(* CODESYS project OC_Core.library
   DefaultNamespace: OC_Core
   DocFormat: reStructuredText
   Description: Open Commissioning TwinCAT Core Library
   Author: SpiraTec AG
   Title: OC_Core
   Version: 1.3.1
   Company: Open Commissioning
   Placeholder: OC_Core

Project tree, tasks and I/O mapping:
  libraries: Tc2_Math, 3.4.4.0 (Beckhoff Automation GmbH); Tc2_Standard, 3.4.5.0 (Beckhoff Automation GmbH); Tc2_System, 3.6.4.0 (Beckhoff Automation GmbH); Tc2_Utilities, 3.6.1.0 (Beckhoff Automation GmbH); Tc3_Module, 3.4.5.0 (Beckhoff Automation GmbH); TcUnit, 1.3.0.0 (www.tcunit.org)
  Common/
    AdsMessageHandler/
      function block FB_AdsMessageHandler [ST]: bIsAdsMessageReadValid, bIsAdsMessageWriteValid, CreateAdsReadMessage, CreateAdsWriteMessage, LogAdsMessage, SendReadResponse, SendWriteResponse, stAdsMessageRead, stAdsMessageWrite
      data type ST_AdsMessage
    Components/
      Encoder/
        function block FB_Encoder [ST]: ControlLogic, INC_TO_LREAL, InitRun, LREAL_TO_INC, SetActualValue
        data type ST_Encoder_Config
      function block FB_Clock [ST]
      function block FB_ClockAdvanced [ST]
      function block FB_DriveControl [ST]: bIsMoving, bIsPositionReached, fAccMax, fPosition, fPositionLimitMax, fPositionLimitMin, fTolerance, fVelocity, MoveAbsolute, MoveVelocity, Stop
      function block FB_Heater [ST]: fValue, InitRun
      function block FB_MoveAbsolute [ST]: bIsReached, fPosition, fVelocity
      function block FB_MoveVelocity [ST]: bIsReached, fAcc, fVelocity
      function block FB_Ping [ST]: InitRun
    FileIo/
      data type E_FileIoState
      function block FB_FileIO [ST]: nBytesRead, nErrorId, Read, sNetId, Write
    Links/
      function block FB_LinkDataByte [ST]: GetLinkControlData, SetLinkStatusData
      function block FB_LinkDataDWord [ST]: GetLinkControlData, SetLinkStatusData
      function block FB_LinkDataLWord [ST]: GetLinkControlData, SetLinkStatusData
      function block FB_LinkDataReal [ST]: GetLinkControlData, SetLinkStatusData
      function block FB_LinkDataWord [ST]: GetLinkControlData, SetLinkStatusData
      function block FB_LinkDevice [ST]: GetControl, SetStatus
    RecordData/
      function block FB_RecordData [ST]: CmpIGrp, CmpInvokeId, CmpIOffs, DataValid, FB_init, GetReadIndication, GetWriteIndication, SendReadResponse, SendWriteResponse, Subscribe
      interface I_RecordData: GetReadIndication, GetWriteIndication, SendReadResponse, SendWriteResponse, Subscribe
      data type ST_RecordIdent
    System/
      data type E_ControllerType
      function F_IsSystemValid [ST]
      function F_LogError [ST]
      function F_LogMessage [ST]
      function F_LogWarning [ST]
      function block FB_Base [ST]
      function block FB_System [ST]: bDebug, bVerbose, eControllerType, fDeltaTime, fTimeScaling, InitRun
      global variables GVL_Core
    Utils/
      data type E_NetworkByteOrder
      function F_Clamp01 [ST]
      function F_Compare [ST]
      function F_GetHByte [ST]
      function F_GetLByte [ST]
      function F_InverBytesOrder [ST]
      function F_Memcpy [ST]
      function F_Norm [ST]
      function F_ScaleLREAL [ST]
      function F_Sign [ST]
      data type ST_ScaleConfig
  Devices/
    Basic/
      function block FB_Button [ST]
      function block FB_Cylinder [ST]
      function block FB_Device [ST]
      function block FB_DeviceByte [ST]
      function block FB_DeviceDWord [ST]
      function block FB_DeviceLWord [ST]
      function block FB_DeviceReal [ST]
      function block FB_DeviceWord [ST]
      function block FB_Drive [ST]
      function block FB_Lamp [ST]
      function block FB_Lock [ST]
      function block FB_Panel [ST]
      function block FB_Reader [ST]
      function block FB_Robot [ST]: ConnectJoints, GetJointsTarget, SetJointsStatus
      function block FB_SensorAnalog [ST]
      function block FB_SensorBinary [ST]
      function block FB_Switch [ST]
*)

// Common/AdsMessageHandler/ST_AdsMessage
TYPE ST_AdsMessage :
STRUCT
	tNetID			: T_AmsNetID; // AMS NetId identifier
	tPort			: T_AmsPort; // AMS port number
	nInvokeID		: UDINT; // Unique identifier for the ADS invocation
	nIdxGrp			: UDINT; // Index group for the ADS command
	nIdxOffs		: UDINT; // Index offset within the ADS command
	nLength			: UDINT; // Length of the ADS message data
	nResult			: UDINT; // Result code from the ADS operation
	aData			: ARRAY[0..239] OF BYTE; // Data payload (240-byte buffer)
END_STRUCT
END_TYPE

// Common/Components/Encoder/ST_Encoder_Config
TYPE ST_Encoder_Config :
STRUCT
	bIsIntegrator   		: BOOL := FALSE;  //Integrate input value
	fNumerator 	  			: REAL := 0.0001; //[unit/INC]
	fDenominator  			: REAL := 1.0; 	// Scaling
	fModulo 	  			: REAL := 0; // Modulo [unit]; If 0, will be ignored
	fGearFactor  			: REAL := 1.0;
	bInvertEncoderDirection : BOOL;
END_STRUCT
END_TYPE

// Common/FileIo/E_FileIoState
{attribute 'conditionalshow'}
TYPE E_FileIoState :
(
	READY := 0,
	OPEN,
	CREATE,
	READ,
	WRITE,
	CLOSE,
	ERROR
);
END_TYPE

// Common/RecordData/ST_RecordIdent
TYPE ST_RecordIdent :
STRUCT
	nPort  			: T_AmsPort; //ADS-Port of the Profinet Device. Ignored when using PLCSIM Advanced
	nSlot			: UINT; //Slotnumber of the Profinet Device. Ignored when using PLCSIM Advanced
	nSubSlot		: UINT; //Subslotnumber of the Profinet Device. Ignored when using PLCSIM Advanced
	nPlcId			: UINT; //Identifier of the PLC when using PLCSIM Advanced
	nHardwareId		: UINT; //Hardware-ID of the device when using PLCSIM Advanced
END_STRUCT
END_TYPE

// Common/System/E_ControllerType
{attribute 'qualified_only'}
{attribute 'strict'}
TYPE E_ControllerType :
(
	NotDefined := 0,
	PlcSimAdvanced := 1
);
END_TYPE

// Common/Utils/E_NetworkByteOrder
{attribute 'qualified_only'}
{attribute 'strict'}
TYPE E_NetworkByteOrder :
(
	BigEndian := 0, //Big Endian (MOTOROLA)
	LittleEndian := 1 //Little Endian (Intel)	
);
END_TYPE

// Common/Utils/ST_ScaleConfig
{attribute 'pack_mode' := '0'} 
TYPE ST_ScaleConfig :
STRUCT
	fInputMin 	: LREAL := 0;
	fInputMax 	: LREAL := 100;
	fOutputMin 	: LREAL := 0;
	fOutputMax 	: LREAL := 65535;
END_STRUCT
END_TYPE

// Common/System/GVL_Core
{attribute 'qualified_only'}
{attribute 'conditionalshow'}
VAR_GLOBAL	
	refSystem 			: REFERENCE TO FB_System;		
END_VAR

// Common/AdsMessageHandler/FB_AdsMessageHandler
(*ADS Message Handler is responsible for indication of the ADS Read/Write messages for local NetId and generation of the response message*)
FUNCTION_BLOCK FB_AdsMessageHandler
VAR_INPUT
	bDisable 				: BOOL;	//Deactivate cyclical execution
	bLog					: BOOL;	//Log ADS messages data in the console
	bVerbose				: BOOL; //Log Verbose information in the console
END_VAR

VAR	
	_fbAdsWriteIndicator 	: AdsWriteInd;	
	_fbAdsReadIndicator 	: AdsReadInd;
	_fbAdsWriteResponse		: AdsWriteRes;
	_fbAdsReadResponse		: AdsReadRes;	
	_stAdsMessageWrite		: ST_AdsMessage;
	_stAdsMessageRead		: ST_AdsMessage;
END_VAR

VAR CONSTANT
	S_FORMAT_RECEIVEWRITE	: STRING := 'AdsWriteInd Port: %X, IdxGrp: %X, IdxOffs: %X, InvokeId %X, Length: %X';
	S_FORMAT_RECEIVEREAD	: STRING := 'AdsReadInd Port: %X, IdxGrp: %X, IdxOffs: %X, InvokeId %X, Length: %X';
	S_FORMAT_RESPONSEWRITE	: STRING := 'AdsWriteRes Port: %X, IdxGrp: %X, IdxOffs: %X, InvokeId %X, Length: %X';
	S_FORMAT_RESPONSEREAD	: STRING := 'AdsReadRes Port: %X, IdxGrp: %X, IdxOffs: %X, InvokeId %X, Length: %X';  
END_VAR

IF bDisable THEN RETURN; END_IF

//Reset Indication and Result FBs
_fbAdsWriteResponse(RESPOND := FALSE);
_fbAdsReadResponse(RESPOND := FALSE);

//Capture all Write requests
_fbAdsWriteIndicator();
CreateAdsWriteMessage();
		
//Capture all Read requests
_fbAdsReadIndicator();
CreateAdsReadMessage();

(*Returns the status of the indication of the read message in the current frame*)
PROPERTY PUBLIC bIsAdsMessageReadValid : BOOL
GET
bIsAdsMessageReadValid := _stAdsMessageRead.tPort <> 0;
END_GET
END_PROPERTY

(*Returns the status of the indication of the write message in the current frame*)
PROPERTY PUBLIC bIsAdsMessageWriteValid : BOOL
GET
bIsAdsMessageWriteValid := _stAdsMessageWrite.tPort <> 0;
END_GET
END_PROPERTY

METHOD PRIVATE CreateAdsReadMessage : BOOL
IF NOT _fbAdsReadIndicator.VALID THEN RETURN; END_IF

MEMSET(ADR(_stAdsMessageRead), 0, SIZEOF(ST_AdsMessage));
_stAdsMessageRead.tNetId 		:= _fbAdsReadIndicator.NETID;
_stAdsMessageRead.tPort 		:= _fbAdsReadIndicator.PORT;
_stAdsMessageRead.nInvokeId 	:= _fbAdsReadIndicator.INVOKEID;
_stAdsMessageRead.nIdxGrp 		:= _fbAdsReadIndicator.IDXGRP;
_stAdsMessageRead.nIdxOffs 		:= _fbAdsReadIndicator.IDXOFFS;
_stAdsMessageRead.nLength 		:= _fbAdsReadIndicator.LENGTH;

IF bVerbose THEN
	LogAdsMessage(_stAdsMessageWrite, S_FORMAT_RECEIVEREAD);
END_IF

_fbAdsReadIndicator(CLEAR := TRUE);
_fbAdsReadIndicator(CLEAR := FALSE);
END_METHOD

METHOD PRIVATE CreateAdsWriteMessage : BOOL
IF NOT _fbAdsWriteIndicator.VALID THEN RETURN; END_IF

MEMSET(ADR(_stAdsMessageWrite), 0, SIZEOF(ST_AdsMessage));
_stAdsMessageWrite.tNetId 		:= _fbAdsWriteIndicator.NETID;
_stAdsMessageWrite.tPort 		:= _fbAdsWriteIndicator.PORT;
_stAdsMessageWrite.nInvokeId 	:= _fbAdsWriteIndicator.INVOKEID;
_stAdsMessageWrite.nIdxGrp 		:= _fbAdsWriteIndicator.IDXGRP;
_stAdsMessageWrite.nIdxOffs 	:= _fbAdsWriteIndicator.IDXOFFS;
_stAdsMessageWrite.nLength 		:= _fbAdsWriteIndicator.LENGTH;
			
//Limit size to 240
IF _stAdsMessageWrite.nLength > 240 THEN
	IF bVerbose THEN
		F_LOGWARNING(CONCAT('WRREC data length limited to 240. Requested data length was ', TO_STRING(_stAdsMessageWrite.nLength)));
	END_IF
	_stAdsMessageWrite.nLength := 240;
END_IF

MEMCPY(ADR(_stAdsMessageWrite.aData), _fbAdsWriteIndicator.DATAADDR, _stAdsMessageWrite.nLength);

IF bVerbose THEN
	LogAdsMessage(_stAdsMessageWrite, S_FORMAT_RECEIVEWRITE);
END_IF

_fbAdsWriteIndicator(CLEAR := TRUE);
_fbAdsWriteIndicator(CLEAR := FALSE);
END_METHOD

METHOD PRIVATE LogAdsMessage : BOOL
VAR_INPUT
	stAdsMessage 			: ST_AdsMessage;
	sFormat 				: STRING;
END_VAR

VAR
	fbFormatString			: FB_FormatString2;
	sMessage				: STRING;
END_VAR
fbFormatString(
	pFormatString := ADR(sFormat),
	arg1 := F_UINT(stAdsMessage.tPort),
	arg2 := F_UDINT(stAdsMessage.nIdxGrp),
	arg3 := F_UDINT(stAdsMessage.nIdxOffs),		
	arg4 := F_UDINT(stAdsMessage.nInvokeID),
	arg5 := F_UDINT(stAdsMessage.nLength),
	pDstString := ADR(sMessage),
	nDstSize := SIZEOF(sMessage));
F_LogMessage(sMessage);
END_METHOD

(*Send ADS Read Response message*)
METHOD PUBLIC SendReadResponse : HRESULT
VAR_INPUT
	stAdsMessage 	: ST_AdsMessage; //Response ADS Message
END_VAR
IF _fbAdsReadResponse.RESPOND THEN
	SendReadResponse := S_PENDING;
	RETURN;
END_IF

//Limit size to 240
IF stAdsMessage.nLength > 240 THEN
	IF bVerbose THEN
		F_LOGWARNING(CONCAT('RDRES data length limited to 240. Requested data length was ', TO_STRING(stAdsMessage.nLength)));
	END_IF
	stAdsMessage.nLength := 240;
END_IF

_fbAdsReadResponse(
	NETID:= stAdsMessage.tNetId, 
	PORT:= stAdsMessage.tPort, 
	INVOKEID:= stAdsMessage.nInvokeId, 
	RESULT:= stAdsMessage.nResult, 
	LEN:= stAdsMessage.nLength,
	DATAADDR:= ADR(stAdsMessage.aData),
	RESPOND:= TRUE);
IF bVerbose OR bLog THEN	
	LogAdsMessage(stAdsMessage, S_FORMAT_RESPONSEREAD);
END_IF

SendReadResponse := S_OK;
END_METHOD

(*Send ADS Write Response message*)
METHOD PUBLIC SendWriteResponse : HRESULT
VAR_INPUT
	stAdsMessage 	: ST_AdsMessage; //Response ADS Message
END_VAR
IF _fbAdsWriteResponse.RESPOND THEN
	SendWriteResponse := S_PENDING;
	RETURN;
END_IF

_fbAdsWriteResponse(
	NETID:= stAdsMessage.tNetId, 
	PORT:= stAdsMessage.tPort, 
	INVOKEID:= stAdsMessage.nInvokeId, 
	RESULT:= stAdsMessage.nResult, 
	RESPOND:= TRUE);	

IF bVerbose OR bLog THEN		
	LogAdsMessage(stAdsMessage, S_FORMAT_RESPONSEWRITE);
END_IF
	
SendWriteResponse := S_OK;
END_METHOD

(*Get last valid ADS Read Message*)
PROPERTY stAdsMessageRead : REFERENCE TO ST_AdsMessage
GET
stAdsMessageRead REF= _stAdsMessageRead;
END_GET
END_PROPERTY

(*Get last valid ADS Write Message*)
PROPERTY stAdsMessageWrite : REFERENCE TO ST_AdsMessage
GET
stAdsMessageWrite REF= _stAdsMessageWrite;
END_GET
END_PROPERTY

END_FUNCTION_BLOCK

// Common/System/F_LogWarning
(*
	Log Warning message to TwinCAT console
*)
{attribute 'hide_all_locals'}
FUNCTION F_LogWarning : BOOL
VAR_INPUT
	sMessage : T_MAXSTRING;
END_VAR

VAR CONSTANT	
	S_LOGHEADER		: T_MAXSTRING := 'Open Commissioning: %s';
END_VAR

ADSLOGSTR(ADSLOG_MSGTYPE_WARN, S_LOGHEADER, sMessage);

END_FUNCTION

// Common/System/F_LogMessage
(*
	Log message to TwinCAT console
*)
{attribute 'hide_all_locals'}
FUNCTION F_LogMessage : BOOL
VAR_INPUT
	sMessage : T_MAXSTRING;
END_VAR

VAR CONSTANT	
	S_LOGHEADER		: T_MAXSTRING := 'Open Commissioning: %s';
END_VAR

ADSLOGSTR(ADSLOG_MSGTYPE_HINT, S_LOGHEADER, sMessage);

END_FUNCTION

// Common/Components/Encoder/FB_Encoder
(*
	Generic simulated Encoder 
*)
{attribute 'reflection'} 
FUNCTION_BLOCK FB_Encoder
VAR_INPUT
	fValue 			: LREAL; //Input Value [unit] or [unit/s]	
	stConfig 		: ST_Encoder_Config;	
END_VAR

VAR_OUTPUT
	nResult 		: DINT; //Position [INC]
	fResult 		: LREAL;
END_VAR

VAR
	{attribute 'instance-path'} 
    {attribute 'noinit'} 
    _sPath 				: STRING;
	_fValue 			: LREAL;
END_VAR

InitRun();
ControlLogic();

METHOD PRIVATE ControlLogic
IF stConfig.bIsIntegrator THEN
	_fValue := _fValue + (fValue * stConfig.fGearFactor * GVL_Core.fbSystem.fDeltaTime);
ELSE
	_fValue := fValue * stConfig.fGearFactor;
END_IF

IF stConfig.fModulo > 0.0 THEN
	_fValue := LREAL_TO_REAL(LMOD(_fValue, stConfig.fModulo));
END_IF

fResult := _fValue;

IF stConfig.bInvertEncoderDirection THEN
	nResult := LREAL_TO_INC(fResult, -1);
ELSE
	nResult := LREAL_TO_INC(fResult, 1);	
END_IF
END_METHOD

METHOD INC_TO_LREAL : LREAL
VAR_INPUT
	nValue : DINT;
	fFactor : LREAL;
END_VAR
//Parameters validation
stConfig.fNumerator := MAX(1E-6, stConfig.fNumerator);
stConfig.fDenominator := MAX(1E-6, stConfig.fDenominator);

INC_TO_LREAL := DINT_TO_REAL(nValue) * (stConfig.fNumerator / stConfig.fDenominator) * fFactor;
END_METHOD

METHOD PRIVATE InitRun
VAR_INST
	bInitRun : BOOL := TRUE;
END_VAR
IF NOT bInitRun THEN RETURN; END_IF
bInitRun := FALSE;
END_METHOD

METHOD LREAL_TO_INC : DINT
VAR_INPUT
	fValue : LREAL;
	fFactor : LREAL;
END_VAR
//Parameters validation
stConfig.fNumerator := MAX(1E-6, stConfig.fNumerator);
stConfig.fDenominator := MAX(1E-6, stConfig.fDenominator);

LREAL_TO_INC := LREAL_TO_DINT(fValue * (stConfig.fDenominator / stConfig.fNumerator) * fFactor);
END_METHOD

METHOD PUBLIC SetActualValue : BOOL
VAR_INPUT
	fValue : LREAL;
END_VAR
_fValue := fValue;
END_METHOD

END_FUNCTION_BLOCK

// Common/Components/FB_Clock
FUNCTION_BLOCK FB_Clock
VAR_INPUT
	tPT		: TIME;
END_VAR

VAR_OUTPUT
	bQ		: BOOL;
END_VAR

VAR
	_fbTon1	: TON;
	_fbTon2	: TON;
END_VAR

_fbTon1.PT := tPT;
_fbTon2.PT := tPT;

_fbTon1(IN := NOT bQ);
_fbTon2(IN := bQ);

IF _fbTon1.Q THEN
	bQ := TRUE;
END_IF

IF _fbTon2.Q THEN
	bQ := FALSE;
END_IF

END_FUNCTION_BLOCK

// Common/Components/FB_ClockAdvanced
FUNCTION_BLOCK FB_ClockAdvanced
VAR_INPUT
	bEnable				: BOOL;
	tImpulsePTHigh		: TIME;
	tImpulsePTLow		: TIME;
	tDelay				: TIME;
	bInvert				: BOOL;
END_VAR

VAR_OUTPUT
	bQ					: BOOL;
END_VAR

VAR
	_fbTon1				: TON;
	_fbTon2				: TON;
	_fbTonDelay 		: TON;
	_bValue 			: BOOL;
END_VAR

_fbTonDelay.IN := bEnable;
_fbTonDelay.PT := tDelay;
_fbTonDelay();

IF NOT bEnable THEN
	bQ := FALSE;
	_fbTon1(IN := FALSE);
	_fbTon2(IN := FALSE);
	RETURN;
END_IF

IF _fbTonDelay.Q THEN
	IF bInvert THEN
		_fbTon1.PT := tImpulsePTHigh;
		_fbTon2.PT := tImpulsePTLow;
	ELSE
		_fbTon1.PT := tImpulsePTLow;
		_fbTon2.PT := tImpulsePTHigh;
	END_IF
	
	_fbTon1(IN := NOT _bValue);
	_fbTon2(IN := _bValue);
	
	IF _fbTon1.Q THEN
		_bValue := TRUE;
	END_IF
	
	IF _fbTon2.Q THEN
		_bValue := FALSE;
	END_IF	
	
	IF bInvert THEN
		bQ := NOT _bValue;
	ELSE
		bQ := _bValue;	
	END_IF	
END_IF

END_FUNCTION_BLOCK

// Common/Components/FB_DriveControl
(*
	FB_DriveControl manages drive operations by integrating absolute position and velocity control.
    It encapsulates the functionalities of FB_MoveAbsolute for absolute movement and FB_MoveVelocity
    for velocity-based control.
*)
FUNCTION_BLOCK FB_DriveControl
VAR
	_fbMoveAbsolute 		: FB_MoveAbsolute();
	_fbMoveVelocity			: FB_MoveVelocity();

	_fPosition 				: REAL;
	_fVelocity 				: REAL;		
	_bIsPositionReached 	: BOOL := TRUE;		
	
	_fPositionLimitMin 		: REAL := -1E+12;
	_fPositionLimitMax 		: REAL := 1E+12;
	_fAccMax				: REAL := 1E+12;	
	_fTolerance				: REAL := 1E-6;	
END_VAR

(*
    Indicates whether the drive is currently in motion.

    The bIsMoving property returns TRUE if the drive is actively moving toward its target.
*)
PROPERTY bIsMoving : BOOL
GET
bIsMoving := NOT F_Compare(_fVelocity, 0, 1E-3);
END_GET
END_PROPERTY

(*
    Indicates whether the drive has reached its target position.

    This property reflects the internal state of the drive control system.
    It returns TRUE if the drive has achieved the desired position within the specified
    tolerance limits; otherwise, it returns FALSE.
*)
PROPERTY bIsPositionReached : BOOL
GET
bIsPositionReached := _bIsPositionReached;
END_GET
END_PROPERTY

(*
    Maximum Acceleration Limit

    The fAccMax property represents the maximum acceleration permitted for drive movements.
*)
PROPERTY fAccMax : REAL
GET
fAccMax := _fAccMax;
END_GET
SET
_fAccMax := fAccMax;
END_SET
END_PROPERTY

(*
    Actual Drive Position
	
	The fPosition property provides the current position for the drive.
*)
PROPERTY fPosition : REAL
GET
fPosition := _fPosition;
END_GET
SET
_fPosition := fPosition;
END_SET
END_PROPERTY

(*
    Maximum Position Limit
	
	The fPositionLimitMax property defines the upper boundary for the drive's position.
*)
PROPERTY fPositionLimitMax : REAL
GET
fPositionLimitMax := _fPositionLimitMax;
END_GET
SET
_fPositionLimitMax := fPositionLimitMax;
END_SET
END_PROPERTY

(*
    Minimum  Position Limit
	
	The fPositionLimitMax property defines the lower boundary for the drive's position.
*)
PROPERTY fPositionLimitMin : REAL
GET
fPositionLimitMin := _fPositionLimitMin;
END_GET
SET
_fPositionLimitMin := fPositionLimitMin;
END_SET
END_PROPERTY

(*
    Position Tolerance
	
	The fTolerance property defines the acceptable error range for the drive's position.
*)
PROPERTY fTolerance : REAL
GET
fTolerance := _fTolerance;
END_GET
SET
_fTolerance := fTolerance;
END_SET
END_PROPERTY

(*
    Actual Drive Velocity
	
	The fVelocity property provides the current velocity for the drive.
*)
PROPERTY fVelocity : REAL
GET
fVelocity := _fVelocity;
END_GET
SET
_fVelocity := fVelocity;
END_SET
END_PROPERTY

(* 
    Moves the drive to an absolute position.
    
    The MoveAbsolute method commands the drive to move to a specified absolute position with a given velocity,
    acceleration, and deceleration.
*)
METHOD MoveAbsolute
VAR_INPUT
	fPosition 			: REAL;
	fVelocity			: REAL;
	fAcceleration		: REAL;
	fDeceleration   	: REAL;
END_VAR
_fbMoveAbsolute.fPosition := _fPosition;
_fbMoveAbsolute.fVelocity := _fVelocity;

_fbMoveAbsolute(
	fTargetPosition := LIMIT(_fPositionLimitMin, fPosition, _fPositionLimitMax),
	fTargetVelocity := fVelocity,
	fAccMax := fAcceleration,
	fDecMax := fDeceleration,
	fTolerance := _fTolerance);					

_fVelocity := _fbMoveAbsolute.fVelocity;
_fPosition := _fbMoveAbsolute.fPosition;

_bIsPositionReached := F_Compare(fPosition, _fPosition, _fTolerance);
END_METHOD

(* 
    Moves the drive using velocity control.
    
    The MoveVelocity method commands the drive to move with a specified velocity and controls the acceleration
    and deceleration parameters. It also enforces position limits to prevent the drive from exceeding its boundaries.
*)
METHOD MoveVelocity
VAR_INPUT
	fVelocity 			: REAL;
	fAcceleration 		: REAL;
	fDeceleration 		: REAL;
END_VAR
_fbMoveVelocity.fVelocity := _fVelocity;
_fbMoveVelocity.fTargetVelocity := fVelocity;
_fbMoveVelocity.fAccMax := fAcceleration;
_fbMoveVelocity.fDecMax := fDeceleration;	
	
IF _fPositionLimitMax <> 0 AND _fPositionLimitMin <> 0 THEN
	IF _fPosition >= _fPositionLimitMax OR _fPosition <= _fPositionLimitMin THEN
		_fbMoveVelocity.fTargetVelocity := 0;
		_fbMoveVelocity.fAccMax := _fAccMax;
		_fbMoveVelocity.fDecMax := _fAccMax;
	END_IF		
END_IF
	
_fbMoveVelocity();
	
_fVelocity := _fbMoveVelocity.fVelocity;	

_fPosition := _fPosition + _fVelocity * GVL_Core.fbSystem.fDeltaTime * GVL_Core.fbSystem.fTimeScaling;
_bIsPositionReached := F_Compare(fPosition, _fPosition, _fTolerance);
END_METHOD

(* 
    Stops the drive movement.
    
    The Stop method decelerates the drive until it comes to a complete halt using the specified deceleration.
*)
METHOD Stop
VAR_INPUT
	fDeceleration 	: REAL; 
END_VAR

VAR
	fSign 			: REAL;
	fAbsVelocity 	: REAL;
END_VAR
fSign := F_Sign(_fVelocity);
fAbsVelocity := ABS(_fVelocity);

IF fAbsVelocity > fTolerance THEN
	fAbsVelocity := fAbsVelocity - ABS(fDeceleration) * GVL_Core.fbSystem.fDeltaTime * GVL_Core.fbSystem.fTimeScaling;
	fAbsVelocity := LIMIT(0, fAbsVelocity, 3.402823E+38);
	_fVelocity := fAbsVelocity * fSign;	
ELSE
	_fVelocity := 0;
END_IF
END_METHOD

END_FUNCTION_BLOCK

// Common/Components/FB_MoveAbsolute
(* 
	FB_MoveAbsolute: Controls absolute movement using target position, velocity, acceleration, and deceleration. 
*)
FUNCTION_BLOCK FB_MoveAbsolute 
VAR_INPUT
	fTargetPosition 	: REAL;
	fTargetVelocity 	: REAL; 
	fAccMax 			: REAL; 
	fDecMax 			: REAL;	
	fTolerance			: REAL := 1E-6;	
END_VAR

VAR
	_fVelocity 			: REAL;
	_fPosition 			: REAL;
	_bIsReached			: BOOL;
END_VAR

fTargetVelocity := ABS(fTargetVelocity); 
fAccMax := ABS(fAccMax);
fDecMax := -ABS(fDecMax);

IF F_Compare(fTargetPosition, _fPosition, fTolerance) THEN
	_fVelocity := 0;
	_fPosition := fTargetPosition;
	_bIsReached := TRUE;	
ELSE
	(* Calculate velocity and position *)
	IF fTargetPosition > _fPosition THEN		
		IF _fVelocity < 0 THEN
			_fVelocity := MIN(_fVelocity - fDecMax * GVL_Core.fbSystem.fDeltaTime * GVL_Core.fbSystem.fTimeScaling, fTargetVelocity);
		ELSE
			IF _fVelocity > fTargetVelocity THEN
				_fVelocity := MAX(_fVelocity + fDecMax * GVL_Core.fbSystem.fDeltaTime * GVL_Core.fbSystem.fTimeScaling, fTargetVelocity);
			ELSE
				_fVelocity := MIN(_fVelocity + fAccMax * GVL_Core.fbSystem.fDeltaTime * GVL_Core.fbSystem.fTimeScaling, fTargetVelocity);
			END_IF

			_fVelocity := MIN(SQRT((_fPosition - fTargetPosition) * 2.0 * fDecMax - 1.5 * GVL_Core.fbSystem.fDeltaTime * GVL_Core.fbSystem.fTimeScaling * fDecMax), _fVelocity);
		END_IF

		_fPosition := _fPosition + MIN(_fVelocity * GVL_Core.fbSystem.fDeltaTime * GVL_Core.fbSystem.fTimeScaling, fTargetPosition - _fPosition);	
	ELSE		
		IF _fVelocity > 0 THEN
			_fVelocity := MAX(_fVelocity + fDecMax * GVL_Core.fbSystem.fDeltaTime * GVL_Core.fbSystem.fTimeScaling, -fTargetVelocity);
		ELSE
			IF _fVelocity < -fTargetVelocity THEN
				_fVelocity := MIN(_fVelocity - fDecMax * GVL_Core.fbSystem.fDeltaTime * GVL_Core.fbSystem.fTimeScaling, -fTargetVelocity);
			ELSE				
				_fVelocity := MAX(_fVelocity - fAccMax * GVL_Core.fbSystem.fDeltaTime * GVL_Core.fbSystem.fTimeScaling, -fTargetVelocity);
			END_IF
			
			_fVelocity := MAX(-SQRT((_fPosition - fTargetPosition) * 2.0 * -fDecMax - 1.5 * GVL_Core.fbSystem.fDeltaTime * GVL_Core.fbSystem.fTimeScaling * fDecMax), _fVelocity);
	   END_IF

		_fPosition := _fPosition + MAX(_fVelocity * GVL_Core.fbSystem.fDeltaTime * GVL_Core.fbSystem.fTimeScaling, fTargetPosition - _fPosition);	
	END_IF;
	
	_bIsReached := FALSE;		
END_IF;

(*
    Indicates whether the drive has reached its target position.

    This property reflects the internal state of the drive control system.
    It returns TRUE if the drive has achieved the desired position within the specified
    tolerance limits; otherwise, it returns FALSE.
*)
PROPERTY bIsReached : BOOL
GET
bIsReached := THIS^._bIsReached;
END_GET
END_PROPERTY

(*
    Actual Drive Position
	
	The fPosition property provides the current position for the drive.
*)
PROPERTY fPosition : REAL
GET
fPosition := _fPosition;
END_GET
SET
_fPosition := fPosition;
END_SET
END_PROPERTY

(*
    Actual Drive Velocity
	
	The fVelocity property provides the current velocity for the drive.
*)
PROPERTY fVelocity : REAL
GET
fVelocity := _fVelocity;
END_GET
SET
_fVelocity := fVelocity;
END_SET
END_PROPERTY

END_FUNCTION_BLOCK

// Common/Utils/F_Compare
(*
	Compare fValueA and fValueB within the specified fTolerance window
*)
{attribute 'hide_all_locals'}
FUNCTION F_Compare : BOOL
VAR_INPUT
	fValueA 		: REAL;
	fValueB 		: REAL;
	fTolerance 		: REAL := 1E-6;	
END_VAR

VAR
	_fDifference 	: REAL;
END_VAR

_fDifference := ABS(fValueB - fValueA);
fTolerance := LIMIT(1E-6, ABS(fTolerance), 1E+6);
F_Compare := fTolerance > _fDifference;

END_FUNCTION

// Common/Components/FB_MoveVelocity
(* 
	FB_MoveVelocity: Adjusts the drive's velocity based on target velocity, acceleration, and deceleration
*)
FUNCTION_BLOCK FB_MoveVelocity
VAR_INPUT
	fTargetVelocity 	: REAL;
	fAccMax 			: REAL;
	fDecMax 			: REAL;
END_VAR

VAR
	_fVelocity 			: REAL;	
	_fAcc 				: REAL;
	_bIsReached			: BOOL;
	_fVelocityTolerance	: REAL;
END_VAR

_bIsReached := FALSE;
IF _fAcc = 0 THEN
	IF ABS(fAccMax) > ABS(fDecMax) THEN
		_fVelocityTolerance := ABS(fAccMax) * GVL_Core.fbSystem.fDeltaTime * GVL_Core.fbSystem.fTimeScaling;
	ELSE
		_fVelocityTolerance := ABS(fDecMax) * GVL_Core.fbSystem.fDeltaTime * GVL_Core.fbSystem.fTimeScaling;
	END_IF
ELSE
	_fVelocityTolerance := ABS(_fAcc) * GVL_Core.fbSystem.fDeltaTime * GVL_Core.fbSystem.fTimeScaling;
END_IF	

(* Calculate acceleration *)
//Hold velocity (velocity reached)
IF F_Compare(fVelocity, fTargetVelocity, _fVelocityTolerance) THEN
	_fAcc := 0;
	_fVelocity := fTargetVelocity;
	_bIsReached := TRUE;
	RETURN;
END_IF

IF _fVelocity - fTargetVelocity > _fVelocityTolerance THEN
	//Decelerate
	IF _fVelocity < 0 THEN
		_fAcc := -ABS(fAccMax);
	ELSE
		_fAcc := -ABS(fDecMax);
	END_IF
 ELSIF _fVelocity - fTargetVelocity < -_fVelocityTolerance THEN
	//Accelerate
	IF _fVelocity < 0 THEN
		_fAcc := ABS(fDecMax);
	ELSE
		_fAcc := ABS(fAccMax);
	END_IF
END_IF

_fVelocity := _fVelocity + _fAcc * GVL_Core.fbSystem.fDeltaTime * GVL_Core.fbSystem.fTimeScaling;
_bIsReached := F_Compare(_fVelocity, fTargetVelocity, _fVelocityTolerance);

(* 
	bIsReached: TRUE if the current velocity has reached the target velocity 
*)
PROPERTY bIsReached : BOOL
GET
bIsReached := THIS^._bIsReached;
END_GET
END_PROPERTY

(*
    Actual Drive Acceleration
	
	The fAcc property provides the current acceleration for the drive.
*)
PROPERTY fAcc : REAL
GET
fAcc := THIS^._fAcc;
END_GET
SET
THIS^._fAcc := fAcc;
END_SET
END_PROPERTY

(*
    Actual Drive Velocity
	
	The fVelocity property provides the current velocity for the drive.
*)
PROPERTY fVelocity : REAL
GET
fVelocity := THIS^._fVelocity;
END_GET
SET
THIS^._fVelocity := fVelocity;
END_SET
END_PROPERTY

END_FUNCTION_BLOCK

// Common/Utils/F_Sign
(*
	Return sign of input value
*)
{attribute 'hide_all_locals'}
FUNCTION F_Sign : REAL
VAR_INPUT
	fValue 	: REAL;
END_VAR

IF (fValue >= 0) THEN
	F_Sign := 1;
ELSE
	F_Sign := -1;	
END_IF

END_FUNCTION

// Common/Components/FB_Heater
FUNCTION_BLOCK FB_Heater
VAR_INPUT
	bEnable 		: BOOL;	
	fHeatingSpeed 	: REAL := 1; //[*/s]
	fCoolingSpeed 	: REAL := 1; //[*/s]
	fLimitMin 		: REAL := 0; //[*]
	fLimitMax 		: REAL := 100; //[*]
END_VAR

VAR_OUTPUT
	bEnabled 		: BOOL;
	bIsLimitMin		: BOOL;
	bIsLimitMax		: BOOL;	
END_VAR

VAR
	_fValue 		: REAL; //[*]
END_VAR

InitRun();

bEnabled := bEnable;

_fValue := _fValue - fCoolingSpeed * GVL_Core.fbSystem.fDeltaTime;

IF bEnable THEN
	_fValue := _fValue + fHeatingSpeed * GVL_Core.fbSystem.fDeltaTime;
END_IF

bIsLimitMin := _fValue <= fLimitMin;
bIsLimitMax := _fValue >= fLimitMax;
_fValue := LIMIT(fLimitMin, _fValue, fLimitMax);

PROPERTY fValue : REAL
GET
fValue := _fValue;
END_GET
SET
_fValue := fValue;
END_SET
END_PROPERTY

METHOD INTERNAL InitRun
VAR_INST
	bInitRun : BOOL := TRUE;
END_VAR
IF NOT bInitRun THEN RETURN; END_IF
bInitRun := FALSE;
END_METHOD

END_FUNCTION_BLOCK

// Common/Components/FB_Ping
(*
	FB for measuring the delay between trigger and feeback signal
	Already in use for measuring the delay between TwinCAT and Unity components
*)

FUNCTION_BLOCK FB_Ping
VAR_INPUT	
	bFeedback 		: BOOL;	// bit from unity status
END_VAR

VAR_OUTPUT
	bTrigger		: BOOL;	// bit to unity control
	nActET			: DWORD;	// elapsed time in ms
	nMaxET			: DWORD;	// max. elapsed time in ms
END_VAR

VAR	
	_bEnable			: BOOL;
	_fbTrigStart		: R_TRIG;
	_fbTrigStop			: R_TRIG;
	_fbTrigRestart 		: F_TRIG;
	_nTimeStart 		: TIME;
	_nTimeStop 			: TIME;
END_VAR

InitRun();

_fbTrigStart(CLK := _bEnable);
_fbTrigStop(CLK := bFeedback);
_fbTrigRestart(CLK := bFeedback);

IF _fbTrigStart.Q OR _fbTrigRestart.Q THEN
	nActET := 0;
	bTrigger := TRUE;
	_nTimeStart := TIME();
END_IF


IF _fbTrigStop.Q THEN
	bTrigger := FALSE;
	_nTimeStop := TIME();
	nActET := TIME_TO_DWORD(_nTimeStop - _nTimeStart);
	IF nActET >= nMaxET THEN
		nMaxET := nActET;
	END_IF
END_IF

METHOD INTERNAL InitRun
VAR_INST
	bInitRun : BOOL := TRUE;
END_VAR
IF NOT bInitRun THEN RETURN; END_IF

bInitRun := FALSE;
nActET := 0;
nMaxET := 0;
END_METHOD

END_FUNCTION_BLOCK

// Common/FileIo/FB_FileIO
(*
	File read/write operations.
*)
FUNCTION_BLOCK FB_FileIO
VAR	
	_sNetId				: STRING;
	_fbFileOpen 		: FB_FileOpen;
	_fbFileWrite 		: FB_FileWrite;
	_fbFileRead 		: FB_FileRead;
	_fbFileClose 		: FB_FileClose;	
	_fbCreateDir		: FB_CreateDir;
	_nHFile 			: UINT := 0;
	_eReadState 		: E_FileIoState := READY;
	_eWriteState 		: E_FileIoState := READY;
	_nBytesReadResult	: UDINT;
	_nErrorIdResult		: UDINT;	
END_VAR

(*
	Number of bytes from last read (maps to _nBytesReadResult)
*)
PROPERTY PUBLIC nBytesRead : UDINT
GET
nBytesRead := _nBytesReadResult;
END_GET
SET
PRIVATE
_nBytesReadResult := nBytesRead;
END_SET
END_PROPERTY

(*
	Last error ID (maps to _nErrorIdResult)
*)
PROPERTY PUBLIC nErrorId : uDINT
GET
nErrorId := _nErrorIdResult;
END_GET
SET
PRIVATE
_nErrorIdResult := nErrorId;
END_SET
END_PROPERTY

(*
	Read data from file
	sFileName (T_MaxString): Name/path of the file to read.
	pData (PVOID): Pointer to the data buffer for storing the file contents.
	nLength (UDINT): Number of bytes to read.
*)
METHOD PUBLIC Read : BOOL
VAR_INPUT
	sFileName	: T_MaxString;	//Name/path of the file to read
	pData		: PVOID;	//ointer to the data buffer for storing the file contents
	nLength		: UDINT; //Number of bytes to read
END_VAR
Read := FALSE;
CASE _eReadState OF
	E_FileIoState.READY:
		_fbFileOpen(sNetId := _sNetId, bExecute := FALSE);
		_fbFileRead(sNetId := _sNetId, bExecute := FALSE);
		_fbFileClose(sNetId := _sNetId, bExecute := FALSE);
		_eReadState := E_FileIoState.OPEN;
		
	E_FileIoState.OPEN:
		nErrorId := 0;
		nBytesRead := 0;
		IF _nHFile = 0 THEN
			_fbFileOpen.sPathName := sFileName;
			_fbFileOpen.nMode := FOPEN_MODEREAD;
			_fbFileOpen.ePath := PATH_GENERIC;
			_fbFileOpen(bExecute := TRUE);
		END_IF
		IF _fbFileOpen.hFile <> 0 AND NOT _fbFileOpen.bBusy AND NOT _fbFileOpen.bError THEN
			_nHFile := _fbFileOpen.hFile;
			_fbFileOpen(bExecute := FALSE);			
			_fbFileRead.hFile := _nHFile;
			_fbFileRead.cbReadLen := nLength;
			_fbFileRead.pReadBuff := pData;
			_eReadState := E_FileIoState.READ;
		END_IF
		IF _fbFileOpen.bError THEN
			_fbFileOpen(bExecute := FALSE);
			nErrorId := _fbFileOpen.nErrId;
			_eReadState := E_FileIoState.CREATE;
		END_IF
		
	E_FileIoState.CREATE:
		IF THIS^.Write(sFileName, pData, nLength) THEN
			IF nErrorId = 0 THEN
				_eReadState := E_FileIoState.OPEN;
			ELSE
				_eReadState := E_FileIoState.ERROR;
			END_IF
		END_IF
				
	E_FileIoState.READ:
		_fbFileRead(bExecute := TRUE);
		IF NOT _fbFileRead.bBusy AND NOT _fbFileRead.bError THEN
			nBytesRead := _fbFileRead.cbRead;
			_fbFileRead(bExecute := FALSE);
			_eReadState := E_FileIoState.CLOSE;
		END_IF
		IF _fbFileRead.bError THEN
			nErrorId := _fbFileRead.nErrId;
			_eReadState := E_FileIoState.ERROR;
		END_IF
		
	E_FileIoState.CLOSE:
		IF _nHFile <> 0 THEN
			_fbFileClose(hFile := _nHFile, bExecute := TRUE);
		END_IF
		IF NOT _fbFileClose.bBusy THEN
			_fbFileClose(bExecute := FALSE);
			_nHFile := 0;
			_eReadState := E_FileIoState.READY;
			Read := TRUE;
		END_IF
				
	E_FileIoState.ERROR:
		F_LogError(CONCAT('Error reading/writing file in ', CONCAT(_sNetId, CONCAT(' - ', sFileName))));
		_eReadState := E_FileIoState.CLOSE;
		
END_CASE
END_METHOD

(*
	Network identifier (maps to _sNetId)
*)
PROPERTY sNetId : STRING
GET
sNetId := _sNetId;
END_GET
SET
_sNetId := sNetId;
END_SET
END_PROPERTY

(*
	Write data to file
	sFileName (T_MaxString): Name/path of the file.
	pData (PVOID): Pointer to the content data buffer.
	nLength (UDINT): Number of bytes to write.
*)
METHOD PUBLIC Write : BOOL
VAR_INPUT
	sFileName	: T_MaxString;	//Name/path of the file
	pData 		: PVOID;	//Pointer to the content data buffer
	nLength 	: UDINT;	//Number of bytes to write
END_VAR
Write := FALSE;
CASE _eWriteState OF
	E_FileIoState.READY:
		_fbFileOpen(sNetId := _sNetId, bExecute := FALSE);
		_fbFileWrite(sNetId := _sNetId, bExecute := FALSE);
		_fbFileClose(sNetId := _sNetId, bExecute := FALSE);
		_fbCreateDir(sNetId := _sNetId, bExecute := FALSE);
		_eWriteState := E_FileIoState.OPEN;
		
	E_FileIoState.OPEN:
		nErrorId := 0;
		IF _nHFile = 0 THEN
			_fbFileOpen.sPathName := sFileName;
			_fbFileOpen.nMode := FOPEN_MODEWRITE;
			_fbFileOpen.ePath := PATH_GENERIC;
			_fbFileOpen(bExecute := TRUE);
		END_IF
		IF _fbFileOpen.hFile <> 0 AND NOT _fbFileOpen.bBusy AND NOT _fbFileOpen.bError THEN
			_nHFile := _fbFileOpen.hFile;
			_fbFileOpen(bExecute := FALSE);					
			_fbFileWrite.hFile := _nHFile;
			_fbFileWrite.cbWriteLen := nLength;
			_fbFileWrite.pWriteBuff := pData;
			_eWriteState := E_FileIoState.WRITE;
		END_IF
		IF _fbFileOpen.bError THEN
			_fbFileOpen(bExecute := FALSE);
			nErrorId := _fbFileOpen.nErrId;
			_eWriteState := E_FileIoState.CREATE;			
		END_IF
		
	E_FileIoState.CREATE:
		_fbCreateDir.sPathName:= sFileName;
		_fbCreateDir.ePath:= PATH_GENERIC;
		_fbCreateDir(bExecute := TRUE);
		IF NOT _fbCreateDir.bBusy AND NOT _fbCreateDir.bError THEN
			nErrorId := 0;
			_fbCreateDir(bExecute := FALSE);
			_eWriteState := E_FileIoState.OPEN;
		END_IF
		IF _fbCreateDir.bError THEN
			nErrorId := _fbCreateDir.nErrId;
			_eWriteState := E_FileIoState.ERROR;			
		END_IF
				
	E_FileIoState.WRITE:
		_fbFileWrite(bExecute := TRUE);
		IF NOT _fbFileWrite.bBusy AND _fbFileWrite.cbWrite = nLength AND NOT _fbFileWrite.bError THEN
			_fbFileWrite(bExecute := FALSE);
			_eWriteState := E_FileIoState.CLOSE;
		END_IF
		IF _fbFileWrite.bError THEN
			nErrorId := _fbFileWrite.nErrId;
			_eWriteState := E_FileIoState.ERROR;
		END_IF
		
	E_FileIoState.CLOSE:
		IF  _nHFile <> 0 THEN
			_fbFileClose(hFile := _nHFile, bExecute := TRUE);
		END_IF
		IF NOT _fbFileClose.bBusy THEN
			_fbFileClose(bExecute := FALSE);
			_nHFile := 0;
			_eWriteState := E_FileIoState.READY;
			Write := TRUE;
		END_IF

	E_FileIoState.ERROR:
		F_LogError(CONCAT('Error reading/writing file in ', CONCAT(_sNetId, CONCAT(' - ', sFileName))));
		_eWriteState := E_FileIoState.CLOSE;	

END_CASE
END_METHOD

END_FUNCTION_BLOCK

// Common/System/F_LogError
(*
	Log Error message to TwinCAT console
*)
{attribute 'hide_all_locals'}
FUNCTION F_LogError : BOOL
VAR_INPUT
	sMessage : T_MAXSTRING;
END_VAR

VAR CONSTANT	
	S_LOGHEADER		: T_MAXSTRING := 'Open Commissioning: %s';
END_VAR

ADSLOGSTR(ADSLOG_MSGTYPE_ERROR, S_LOGHEADER, sMessage);

END_FUNCTION

// Common/Links/FB_LinkDataByte
(*
	Link component with additional interface:
	Control BYTE: From TwinCAT >>> To Unity	(Default)
	Status BYTE: FROM Unity >>> TO TwinCAT	(Default)	
	ControlData BYTE: From TwinCAT >>> To Unity		
	StatusData BYTE: FROM Unity >>> TO TwinCAT	
*)
FUNCTION_BLOCK FB_LinkDataByte EXTENDS FB_LinkDevice
VAR	
	{attribute 'simulation_interface'}
	ControlData		AT %Q* : BYTE;
	{attribute 'simulation_interface'}
	StatusData		AT %I* : BYTE;
END_VAR

SUPER^();

METHOD INTERNAL GetLinkControlData : BYTE
GetLinkControlData := ControlData;
END_METHOD

METHOD INTERNAL SetLinkStatusData : BOOL
VAR_INPUT
	nStatusData : BYTE;
END_VAR
StatusData := nStatusData;
END_METHOD

END_FUNCTION_BLOCK

// Common/Links/FB_LinkDevice
(*
	Base link component with default interface:
	Control BYTE: From TwinCAT >>> To Unity
	Status BYTE: FROM Unity >>> TO TwinCAT		
*)
FUNCTION_BLOCK FB_LinkDevice EXTENDS FB_Base
VAR		
	{attribute 'simulation_interface'}
	Control		AT %Q* : BYTE;
	{attribute 'simulation_interface'}
	Status		AT %I* : BYTE;
END_VAR

SUPER^();

METHOD INTERNAL GetControl : BYTE
GetControl := Control;
END_METHOD

METHOD INTERNAL SetStatus : BOOL
VAR_INPUT
	nStatus : BYTE;
END_VAR
Status := nStatus;
END_METHOD

END_FUNCTION_BLOCK

// Common/System/FB_Base
FUNCTION_BLOCK FB_Base

F_IsSystemValid();

END_FUNCTION_BLOCK

// Common/System/F_IsSystemValid
FUNCTION INTERNAL F_IsSystemValid : BOOL
VAR_STAT
	{attribute 'hide'}
	fbTcConfig		: TC_Config;	
	{attribute 'hide'}
	bIsRequested 	: BOOL;
	{attribute 'hide'}
	bIsSystemValid	: BOOL;
END_VAR

IF NOT bIsRequested THEN
	IF NOT __ISVALIDREF(GVL_Core.refSystem) THEN	
		ADSLOGSTR(msgCtrlMask := ADSLOG_MSGTYPE_ERROR OR ADSLOG_MSGTYPE_MSGBOX, 'OC: %s', 'FB_System can not be found! TwinCAT is switched to Config Mode');
		fbTcConfig(NETID := '', SET := TRUE);
		bIsSystemValid := FALSE;
	ELSE
		bIsSystemValid := TRUE;
	END_IF
END_IF

bIsRequested := TRUE;
F_IsSystemValid := bIsSystemValid;

END_FUNCTION

// Common/System/FB_System
(*
	FB_System should be defined and called up once in the project so that the GVL reference is correctly assigned. 
	If FB_System is not defined or there are several instances, the TwinCAT PLC project is forced into config mode with corresponding messages in the console.
*)
{attribute 'reflection'} 
FUNCTION_BLOCK FB_System
VAR_INPUT
	fbAdsMessageHandler 	: FB_AdsMessageHandler;
	fbRecordData 			: FB_RecordData(refAdsMessageHandler := fbAdsMessageHandler);
END_VAR

VAR
	{attribute 'simulation_interface'}
	Control				AT %Q* : BYTE;
	{attribute 'simulation_interface'}
	Status				AT %I* : BYTE;
	{attribute 'simulation_interface'}
	TimeScaling			AT %I* : REAL := 1.0;
	
	{attribute 'instance-path'} 
    {attribute 'noinit'} 
	_sPath 				: STRING;
	
	_bDebug				: BOOL;
	_bVerbose			: BOOL;
	_fDeltaTime 		: REAL;
	_fTimeScaling 		: REAL;
	_eControllerType	: E_ControllerType;
	
	_fbPing				: FB_Ping;
	
	{attribute 'hide'}
	_fbGetCurTaskIdx 	: TC2_SYSTEM.GETCURTASKINDEX;
END_VAR

InitRun();
fTimeScaling := TimeScaling;
_fbPing(bFeedback := Status.7, bTrigger => Control.7);

fbRecordData(); //Execution order -1 relative to FB_AdsMessageHandler
fbAdsMessageHandler();

PROPERTY bDebug : BOOL
GET
bDebug := _bDebug;
END_GET
SET
_bDebug := bDebug;
END_SET
END_PROPERTY

PROPERTY bVerbose : BOOL
GET
bVerbose := _bVerbose;
END_GET
SET
_bVerbose := bVerbose;
END_SET
END_PROPERTY

PROPERTY eControllerType : E_ControllerType
GET
eControllerType := _eControllerType;
END_GET
SET
_eControllerType := eControllerType;
END_SET
END_PROPERTY

PROPERTY PUBLIC fDeltaTime : REAL
GET
fDeltaTime := _fDeltaTime;
END_GET
SET
PRIVATE
_fDeltaTime := fDeltaTime;
END_SET
END_PROPERTY

PROPERTY PUBLIC fTimeScaling : REAL
GET
fTimeScaling := _fTimeScaling;
END_GET
SET
IF fTimeScaling = 0 THEN
	_fTimeScaling := 1.0;
ELSE
	_fTimeScaling := LIMIT(0.01000001, fTimeScaling, 100.0);	
END_IF
END_SET
END_PROPERTY

METHOD PRIVATE InitRun
VAR_INST
	bInitRun 			: BOOL := TRUE;
	sMessageFormat   	: T_MAXSTRING := '%s %s';
	sMessage  			: T_MAXSTRING;
	fbFormatString 		: FB_FormatString;
END_VAR
IF NOT bInitRun THEN RETURN; END_IF
bInitRun := FALSE;

IF __ISVALIDREF(GVL_Core.refSystem) THEN	
	fbFormatString(sFormat := sMessageFormat, arg1 := F_STRINGEx(_sPath), arg2 := F_STRINGEx('FB_System has no single instance! Check the PROGRAM declaration'), sOut => sMessage);
	ADSLOGSTR(msgCtrlMask := ADSLOG_MSGTYPE_ERROR, '%s', sMessage);	
ELSE 
	GVL_Core.refSystem REF= THIS^;
END_IF

_fbGetCurTaskIdx();
_fDeltaTime := UDINT_TO_REAL(TwinCAT_SystemInfoVarList._TaskInfo[_fbGetCurTaskIdx.index].CycleTime / 10000) / 1000.0;
_fTimeScaling := 1;

fbRecordData.eControllerType := _eControllerType;
END_METHOD

END_FUNCTION_BLOCK

// Common/RecordData/FB_RecordData
(*
	Uses an external ADS message handler (FB_AdsMessageHandler) for sending/receiving ADS messages.
	Handles cyclic execution for processing ADS messages and maintains a list of subscribed devices.	
*)
{attribute 'conditionalshow_all_locals}
FUNCTION_BLOCK PUBLIC FB_RecordData IMPLEMENTS I_RecordData
VAR_INPUT
	bDisable 				: BOOL; //Disables cyclic execution when set to TRUE
	bVerbose 				: BOOL; //Enables console logging of ADS message data
	eControllerType 		: E_ControllerType; //Determines data processing logic based on the controller type
END_VAR

VAR	
	_refAdsMessageHandler	: REFERENCE TO FB_AdsMessageHandler;	//Reference to the external ADS message handler used for managing ADS messages	
	_nDeviceCount			: INT;	//Number of devices subscribed for record data
	_aDeviceList			: ARRAY[0..255] OF UDINT; //The internal device list is used for assistance services. Do not delete or change. 
END_VAR

IF bDisable THEN RETURN; END_IF

//Send WriteRes if last WriteInd has not been read by any device
IF _refAdsMessageHandler.stAdsMessageWrite.tPort <> 0 THEN
	SendWriteResponse(_refAdsMessageHandler.stAdsMessageRead);
	_refAdsMessageHandler.stAdsMessageWrite.tPort := 0;
END_IF

//Send ReadRes if last ReadInd has not been read by any device
IF _refAdsMessageHandler.stAdsMessageRead.tPort <> 0 THEN
	SendReadResponse(_refAdsMessageHandler.stAdsMessageRead);
	_refAdsMessageHandler.stAdsMessageRead.tPort := 0;
END_IF 

(*Ads Message Comments*)
//tNetId			: T_AmsNetID;
//tPort				: T_AmsPort;
//nInvokeId			: UDINT; //Hil: Byte0 and 1 = Port, Byte2 = Subslot, Byte3 = Slot. Sil: ignored.
//nIndexGroup		: UDINT; //16#80000000 + RecordIndex
//nIndexOffset		: UDINT; //Hil: LowWord = SubSlot, HighWord = Slot. Sil: LowWord = HardwareId, HighWord = PlcId.
//nLengthData		: UDINT;
//nResult			: UDINT;
//aData				: ARRAY[0..239] OF BYTE;

METHOD PRIVATE CmpIGrp : BOOL
VAR_INPUT
	nIGrpDevice 	: UDINT;
	nIGrpReceived 	: UDINT;
END_VAR
(* Compare low word only *)
CmpIGrp := (nIGrpDevice AND 16#0000FFFF) = (nIGrpReceived AND 16#0000FFFF) OR nIGrpDevice = 0;
END_METHOD

METHOD PRIVATE CmpInvokeId : BOOL
VAR_INPUT
	nInvokeIdDevice 	: UDINT;
	nInvokeIdReceived 	: UDINT;
END_VAR
IF eControllerType = E_ControllerType.PlcSimAdvanced THEN
	CmpInvokeId := TRUE;
	RETURN;
END_IF

(* Compare low word only. low word = port *)
CmpInvokeId := (nInvokeIdDevice AND 16#0000FFFF) = (nInvokeIdReceived AND 16#0000FFFF);
END_METHOD

METHOD PRIVATE CmpIOffs : BOOL
VAR_INPUT
	nIOffsDevice 	: UDINT;
	nIOffsReceived 	: UDINT;
END_VAR
CmpIOffs := nIOffsDevice = nIOffsReceived OR nIOffsDevice = 16#FFFFFFFF;
END_METHOD

METHOD INTERNAL DataValid : BOOL
VAR_INPUT
	refDeviceAdsMessage 	: REFERENCE TO ST_AdsMessage;
	refHandlerAdsMessage	: REFERENCE TO ST_AdsMessage;
END_VAR
DataValid := FALSE;

IF refHandlerAdsMessage.tPort = 0 THEN
	RETURN;
END_IF

IF NOT CmpInvokeId(refDeviceAdsMessage.nInvokeId, refHandlerAdsMessage.nInvokeId) THEN
	RETURN;
END_IF

IF NOT CmpIOffs(refDeviceAdsMessage.nIdxOffs, refHandlerAdsMessage.nIdxOffs) THEN
	RETURN;
END_IF

IF NOT CmpIGrp(refDeviceAdsMessage.nIdxGrp, refHandlerAdsMessage.nIdxGrp) THEN
	RETURN;
END_IF

(* Copy the received telegram *)
MEMCPY(ADR(refDeviceAdsMessage), ADR(refHandlerAdsMessage), SIZEOF(ST_AdsMessage));

(* Indicate that the telegram has been read by a device
   -> the device is now responsible for the response! *)
refHandlerAdsMessage.tPort := 0;

DataValid := TRUE;
END_METHOD

METHOD FB_init : BOOL
VAR_INPUT
	bInitRetains 				: BOOL; // if TRUE, the retain variables are initialized (warm start / cold start)
	bInCopyCode 				: BOOL;  // if TRUE, the instance afterwards gets moved into the copy code (online change)
	refAdsMessageHandler		: REFERENCE TO FB_AdsMessageHandler;
END_VAR
THIS^._refAdsMessageHandler REF= refAdsMessageHandler;
END_METHOD

(*Try to get a valid ADR read message. If the message is valid, the data in the input structure will be overwritten*)
METHOD PUBLIC GetReadIndication : BOOL
VAR_INPUT
	refDeviceAdsMessage : REFERENCE TO ST_AdsMessage; //Reference ADS Message
END_VAR
IF NOT _refAdsMessageHandler.bIsAdsMessageReadValid THEN
	GetReadIndication := FALSE;
	RETURN; 
END_IF

GetReadIndication := DataValid(refDeviceAdsMessage, _refAdsMessageHandler.stAdsMessageRead);
END_METHOD

(*Try to get a valid ADR write message. If the message is valid, the data in the input structure will be overwritten*)
METHOD PUBLIC GetWriteIndication : BOOL
VAR_INPUT
	refDeviceAdsMessage : REFERENCE TO ST_AdsMessage; //Reference ADS Message	
END_VAR
IF NOT _refAdsMessageHandler.bIsAdsMessageWriteValid THEN
	GetWriteIndication := FALSE;
	RETURN; 
END_IF

GetWriteIndication := DataValid(refDeviceAdsMessage, _refAdsMessageHandler.stAdsMessageWrite);
END_METHOD

(*Send ADS Read Response message*)
METHOD PUBLIC SendReadResponse : HRESULT
VAR_INPUT
	stAdsMessage : ST_AdsMessage; //Response ADS Message
END_VAR
CASE eControllerType OF		
	E_ControllerType.PlcSimAdvanced :
		stAdsMessage.nResult := SHR(stAdsMessage.nIdxOffs, 16) + 16#80000000;
END_CASE

SendReadResponse := _refAdsMessageHandler.SendReadResponse(stAdsMessage);
END_METHOD

(*Send ADS Write Response message*)
METHOD PUBLIC SendWriteResponse : HRESULT
VAR_INPUT
	stAdsMessage : ST_AdsMessage; //Response ADS Message
END_VAR
CASE eControllerType OF		
	E_ControllerType.PlcSimAdvanced :
		stAdsMessage.nResult := SHR(stAdsMessage.nIdxOffs, 16) + 16#80000000;
END_CASE

SendWriteResponse := _refAdsMessageHandler.SendWriteResponse(stAdsMessage);
END_METHOD

(*Subscribe the RecordIdent device to the RecordData services. The RecordIdent device is initialised during subscription*)
METHOD PUBLIC Subscribe
VAR_INPUT
	pRecordIdent	: POINTER TO ST_RecordIdent; //Pointet to RecordIdent Device
	stAdsMessage 	: REFERENCE TO ST_AdsMessage; //Reference to the initial ADS message configuration of the device
END_VAR
IF _nDeviceCount > 255 THEN
	F_LogError('More than 256 RecordData devices');
	RETURN;
END_IF

CASE eControllerType OF
	E_ControllerType.NotDefined :	
		stAdsMessage.nInvokeId := pRecordIdent^.nPort + UINT_TO_USINT(pRecordIdent^.nSubSlot) * 16#10000 + UINT_TO_USINT(pRecordIdent^.nSlot) * 16#1000000;		
		stAdsMessage.nIdxOffs := pRecordIdent^.nSubSlot + pRecordIdent^.nSlot * 16#10000;	
		stAdsMessage.tPort := pRecordIdent^.nPort;
		
		IF stAdsMessage.nInvokeId = 0 THEN
			RETURN;
		END_IF
		
		_aDeviceList[_nDeviceCount] := stAdsMessage.nInvokeId;
	
	E_ControllerType.PlcSimAdvanced :
		stAdsMessage.nIdxOffs := pRecordIdent^.nHardwareId + pRecordIdent^.nPlcId * 16#10000;
		
		IF stAdsMessage.nIdxOffs = 0 THEN
			RETURN;
		END_IF
		
		_aDeviceList[_nDeviceCount] := stAdsMessage.nIdxOffs;
END_CASE	

_nDeviceCount := _nDeviceCount + 1;
END_METHOD

END_FUNCTION_BLOCK

// Common/RecordData/I_RecordData
{attribute 'conditionalshow'}
INTERFACE I_RecordData

(*Try to get a valid ADR read message. If the message is valid, the data in the input structure will be overwritten*)
METHOD GetReadIndication : BOOL
VAR_INPUT
	refDeviceAdsMessage : REFERENCE TO ST_AdsMessage; //Reference ADS Message
END_VAR
END_METHOD

(*Try to get a valid ADR write message. If the message is valid, the data in the input structure will be overwritten*)
METHOD GetWriteIndication : BOOL
VAR_INPUT
	refDeviceAdsMessage : REFERENCE TO ST_AdsMessage; //Reference ADS Message
END_VAR
END_METHOD

(*Send ADS Read Response message*)
METHOD SendReadResponse : HRESULT
VAR_INPUT
	stAdsMessage : ST_AdsMessage; //Response ADS Message
END_VAR
END_METHOD

(*Send ADS Write Response message*)
METHOD SendWriteResponse : HRESULT
VAR_INPUT
	stAdsMessage : ST_AdsMessage; //Response ADS Message
END_VAR
END_METHOD

(*Subscribe the RecordIdent device to the RecordData services. The RecordIdent device is initialised during subscription*)
METHOD Subscribe
VAR_INPUT
	pRecordIdent	: POINTER TO ST_RecordIdent; //Pointet to RecordIdent Device
	stAdsMessage 	: REFERENCE TO ST_AdsMessage; //Reference to the initial ADS message configuration of the device
END_VAR
END_METHOD

END_INTERFACE

// Common/Links/FB_LinkDataDWord
(*
	Link component with additional interface:
	Control BYTE: From TwinCAT >>> To Unity	(Default)
	Status BYTE: FROM Unity >>> TO TwinCAT	(Default)
	ControlData DWORD: From TwinCAT >>> To Unity		
	StatusData DWORD: FROM Unity >>> TO TwinCAT		
*)
FUNCTION_BLOCK FB_LinkDataDWord EXTENDS FB_LinkDevice
VAR		
	{attribute 'simulation_interface'}
	ControlData		AT %Q* : DWORD;
	{attribute 'simulation_interface'}
	StatusData		AT %I* : DWORD;
END_VAR

SUPER^();

METHOD INTERNAL GetLinkControlData : DWORD
GetLinkControlData := ControlData;
END_METHOD

METHOD INTERNAL SetLinkStatusData : BOOL
VAR_INPUT
	nStatusData : DWORD;
END_VAR
StatusData := nStatusData;
END_METHOD

END_FUNCTION_BLOCK

// Common/Links/FB_LinkDataLWord
(*
	Link component with additional interface:
	Control BYTE: From TwinCAT >>> To Unity	(Default)
	Status BYTE: FROM Unity >>> TO TwinCAT	(Default)
	ControlData LWORD: From TwinCAT >>> To Unity		
	StatusData LWORD: FROM Unity >>> TO TwinCAT		
*)
FUNCTION_BLOCK FB_LinkDataLWord EXTENDS FB_LinkDevice
VAR	
	{attribute 'simulation_interface'}
	ControlData		AT %Q* : LWORD;
	{attribute 'simulation_interface'}
	StatusData		AT %I* : LWORD;
END_VAR

SUPER^();

METHOD INTERNAL GetLinkControlData : LWORD
GetLinkControlData := ControlData;
END_METHOD

METHOD INTERNAL SetLinkStatusData : BOOL
VAR_INPUT
	nStatusData : LWORD;
END_VAR
StatusData := nStatusData;
END_METHOD

END_FUNCTION_BLOCK

// Common/Links/FB_LinkDataReal
(*
	Link component with additional interface:
	Control BYTE: From TwinCAT >>> To Unity	(Default)
	Status BYTE: FROM Unity >>> TO TwinCAT	(Default)
	ControlData REAL: From TwinCAT >>> To Unity		
	StatusData REAL: FROM Unity >>> TO TwinCAT		
*)
FUNCTION_BLOCK FB_LinkDataReal EXTENDS FB_LinkDevice
VAR	
	{attribute 'simulation_interface'}
	ControlData			AT %Q* : REAL;
	{attribute 'simulation_interface'}
	StatusData			AT %I* : REAL;
END_VAR

SUPER^();

METHOD INTERNAL GetLinkControlData : REAL
GetLinkControlData := ControlData;
END_METHOD

METHOD INTERNAL SetLinkStatusData : BOOL
VAR_INPUT
	fStatusData : REAL;
END_VAR
StatusData := fStatusData;
END_METHOD

END_FUNCTION_BLOCK

// Common/Links/FB_LinkDataWord
(*
	Link component with additional interface:
	Control BYTE: From TwinCAT >>> To Unity	(Default)
	Status BYTE: FROM Unity >>> TO TwinCAT	(Default)
	ControlData WORD: From TwinCAT >>> To Unity		
	StatusData WORD: FROM Unity >>> TO TwinCAT		
*)
FUNCTION_BLOCK FB_LinkDataWord EXTENDS FB_LinkDevice
VAR	
	{attribute 'simulation_interface'}
	ControlData		AT %Q* : WORD;
	{attribute 'simulation_interface'}
	StatusData		AT %I* : WORD;	
END_VAR

SUPER^();

METHOD INTERNAL GetLinkControlData : WORD
GetLinkControlData := ControlData;
END_METHOD

METHOD INTERNAL SetLinkStatusData : BOOL
VAR_INPUT
	nStatusData : WORD;
END_VAR
StatusData := nStatusData;
END_METHOD

END_FUNCTION_BLOCK

// Common/Utils/F_Clamp01
(*
	Clamp the input value within the range of 0 to 1
*)
FUNCTION F_Clamp01 : REAL
VAR_INPUT
	fValue : REAL;
END_VAR

F_Clamp01:= LIMIT(0, fValue, 1);

END_FUNCTION

// Common/Utils/F_GetHByte
(*
	Return the high byte from the input word
*)
FUNCTION F_GetHByte : BYTE
VAR_INPUT
	nWord	: WORD;
END_VAR

F_GetHByte := WORD_TO_BYTE(SHR(nWord, 8));

END_FUNCTION

// Common/Utils/F_GetLByte
(*
	Return the low byte from the input word
*)
FUNCTION F_GetLByte : BYTE
VAR_INPUT
	nWord	: WORD;
END_VAR

F_GetLByte := WORD_TO_BYTE(nWord);

END_FUNCTION

// Common/Utils/F_InverBytesOrder
(*
	Reverse the byte order of the given ANY input.
*)
FUNCTION F_InverBytesOrder : BOOL
VAR_INPUT
	data 	: ANY;
END_VAR

VAR	
	_i 		: UDINT;
	_nSize	: UDINT;
	_aData 	: ARRAY [0..7] OF BYTE;
END_VAR

_nSize := DINT_TO_UDINT(data.diSize);
MEMCPY(ADR(_aData), data.pValue, _nSize);

IF(_nSize > 8) THEN
	F_LogError('F_InverBytesOrder: Data Size is not in range [0..7]');
	RETURN;
END_IF

FOR _i:= 1 TO _nSize DO	
	MEMCPY(data.pValue + _i - 1, ADR(_aData) + _nSize - _i, 1);
END_FOR

END_FUNCTION

// Common/Utils/F_Memcpy
(*
	Custom MEMCPY function with a swap flag. 
	If bSwap is true and the length is within the range of 0 to 8, the memcpy operation will be performed with reversed byte order.
*) 
FUNCTION F_Memcpy : UDINT
VAR_INPUT
	destAddr 	: PVOID; //Destination Addr
	srcAddr 	: PVOID; //Source Addr
	n			: UDINT; //Bytes Length
	bSwap		: BOOL; //If TRUE and the length is within the range of 0 to 8, the memcpy operation will be performed with reversed byte order
END_VAR

VAR
	i 			: UDINT;
	aBuffer 	: ARRAY [0..7] OF BYTE;
	nWWORD		: WORD;
	nDWORD		: DWORD;
	nLWORD		: LWORD;
END_VAR

IF NOT bSWAP OR n > 8 THEN
	F_MEMCPY := MEMCPY(destAddr, srcAddr, n);
	RETURN;
END_IF

F_MEMCPY := MEMCPY(ADR(aBuffer), srcAddr, n);

FOR i:= 1 TO n DO	
	MEMCPY(destAddr + i - 1, ADR(aBuffer) + n - i, 1);
END_FOR

END_FUNCTION

// Common/Utils/F_Norm
(*
	The input value will be normalized in the range of fMin to fMax.
	The returned value is within the range of 0 to 1.
*)
FUNCTION F_Norm : REAL
VAR_INPUT
	fMin 		: REAL; //Limit Min
	fMax 		: REAL; //Limit Max
	fValue 		: REAL; //Input Value
END_VAR

F_Norm := F_Clamp01((fValue - fMin)/(fMax - fMin));

END_FUNCTION

// Common/Utils/F_ScaleLREAL
(*
 	The input value will be normalize scaled from the input range [fInputMin..fInputMax] to the output range [fOutputMin..fOutputMax].	
*)
FUNCTION F_ScaleLREAL : LREAL
VAR_INPUT
	fValue 		: LREAL; //Input value
	fInputMin 	: LREAL; //Input limit Min
	fInputMax 	: LREAL; //Input limit Max
	fOutputMin 	: LREAL; //Output limit Min
	fOutputMax 	: LREAL; //Output limit Max
END_VAR

VAR
	fNormalized : LREAL;
END_VAR

VAR_OUTPUT
	bError 		: BOOL;
END_VAR

bError := (fInputMin >= fInputMax) OR (fOutputMin >= fOutputMax);

IF bError THEN
	F_ScaleLREAL := 0.0;
	RETURN;
END_IF

IF fValue < fInputMin THEN
	fNormalized := 0.0;
ELSIF fValue > fInputMax THEN
	fNormalized := 1.0;
ELSE
	fNormalized := (fValue - fInputMin) / (fInputMax - fInputMin);
END_IF

F_ScaleLREAL := fNormalized * (fOutputMax - fOutputMin) + fOutputMin;

END_FUNCTION

// Devices/Basic/FB_Button
(*
	Default button device.
*)
FUNCTION_BLOCK FB_Button EXTENDS FB_LinkDevice 
VAR_INPUT
	bEnable		: BOOL; //0-Lamp OFF, 1-Lamp ON
END_VAR

VAR_OUTPUT
	bValue		: BOOL; //0-Released, 1-Pressed
END_VAR

SUPER^();
Control.0 := bEnable;
bValue := Status.0;

END_FUNCTION_BLOCK

// Devices/Basic/FB_Cylinder
(*
	Default cylinder (valve) device.
*)
FUNCTION_BLOCK FB_Cylinder EXTENDS FB_LinkDevice 
VAR_INPUT
	bRetract : BOOL; //Move to MIN
	bExtend : BOOL; //Move to MAX
END_VAR

VAR_OUTPUT
	bRetracted : BOOL; //Is in MIN
	bExtended : BOOL; //Is in MAX
END_VAR

SUPER^();
bRetracted := Status.0;
bExtended := Status.1;
Control.0 := bRetract;
Control.1 := bExtend;

END_FUNCTION_BLOCK

// Devices/Basic/FB_Device
(*
	Basic device with default interface:
	nControl BYTE: From TwinCAT >>> To Unity
	nStatus BYTE: FROM Unity >>> TO TwinCAT		
*)
FUNCTION_BLOCK FB_Device EXTENDS FB_LinkDevice
VAR_INPUT		
	nControl  			: BYTE;
END_VAR

VAR_OUTPUT
	nStatus  			: BYTE;
END_VAR

SUPER^();
Control := nControl;
nStatus := Status;

END_FUNCTION_BLOCK

// Devices/Basic/FB_DeviceByte
(*
	Basic device with extended interface:
	nControl BYTE: From TwinCAT >>> To Unity
	nStatus BYTE: FROM Unity >>> TO TwinCAT	
	nControlData BYTE: From TwinCAT >>> To Unity
	nStatusData BYTE: FROM Unity >>> TO TwinCAT	
*)
FUNCTION_BLOCK FB_DeviceByte EXTENDS FB_LinkDataByte
VAR_INPUT		
	nControl  			: BYTE;
	nControlData  		: BYTE;
END_VAR

VAR_OUTPUT
	nStatus  			: BYTE;
	nStatusData  		: BYTE;
END_VAR

SUPER^();
Control := nControl;
ControlData := nControlData;
nStatus := Status;
nStatusData := StatusData;

END_FUNCTION_BLOCK

// Devices/Basic/FB_DeviceDWord
(*
	Basic device with extended interface:
	nControl BYTE: From TwinCAT >>> To Unity
	nStatus BYTE: FROM Unity >>> TO TwinCAT	
	nControlData DWORD: From TwinCAT >>> To Unity
	nStatusData DWORD: FROM Unity >>> TO TwinCAT	
*)
FUNCTION_BLOCK FB_DeviceDWord EXTENDS FB_LinkDataDWord
VAR_INPUT		
	nControl  			: BYTE;
	nControlData 		: DWORD;
END_VAR

VAR_OUTPUT
	nStatus  			: BYTE;
	nStatusData  		: DWORD;
END_VAR

SUPER^();
Control := nControl;
ControlData := nControlData;
nStatus := Status;
nStatusData := StatusData;

END_FUNCTION_BLOCK

// Devices/Basic/FB_DeviceLWord
(*
	Basic device with extended interface:
	nControl BYTE: From TwinCAT >>> To Unity
	nStatus BYTE: FROM Unity >>> TO TwinCAT	
	nControlData LWORD: From TwinCAT >>> To Unity
	nStatusData LWORD: FROM Unity >>> TO TwinCAT	
*)
FUNCTION_BLOCK FB_DeviceLWord EXTENDS FB_LinkDataLWord
VAR_INPUT		
	nControl  			: BYTE;
	nControlData  		: LWORD;
END_VAR

VAR_OUTPUT
	nStatus  			: BYTE;
	nStatusData  		: LWORD;
END_VAR

SUPER^();
Control := nControl;
ControlData := nControlData;
nStatus := Status;
nStatusData := StatusData;

END_FUNCTION_BLOCK

// Devices/Basic/FB_DeviceReal
(*
	Basic device with extended interface:
	nControl BYTE: From TwinCAT >>> To Unity
	nStatus BYTE: FROM Unity >>> TO TwinCAT	
	fControlData REAL: From TwinCAT >>> To Unity
	fStatusData REAL: FROM Unity >>> TO TwinCAT	
*)
FUNCTION_BLOCK FB_DeviceReal EXTENDS FB_LinkDataReal
VAR_INPUT		
	nControl  			: BYTE;
	fControlData  		: REAL;
END_VAR

VAR_OUTPUT
	nStatus  			: BYTE;
	fStatusData  		: REAL;
END_VAR

SUPER^();
Control := nControl;
ControlData := fControlData;
nStatus := Status;
fStatusData := StatusData;

END_FUNCTION_BLOCK

// Devices/Basic/FB_DeviceWord
(*
	Basic device with extended interface:
	nControl BYTE: From TwinCAT >>> To Unity
	nStatus BYTE: FROM Unity >>> TO TwinCAT	
	nControlData WORD: From TwinCAT >>> To Unity
	nStatusData WORD: FROM Unity >>> TO TwinCAT	
*)
FUNCTION_BLOCK FB_DeviceWord EXTENDS FB_LinkDataWord
VAR_INPUT		
	nControl  			: BYTE;
	nControlData  		: WORD;
END_VAR

VAR_OUTPUT
	nStatus  			: BYTE;
	nStatusData  		: WORD;
END_VAR

SUPER^();
Control := nControl;
ControlData := nControlData;
nStatus := Status;
nStatusData := StatusData;

END_FUNCTION_BLOCK

// Devices/Basic/FB_Drive
(*
	Basic drive interface:
	nControl BYTE: From TwinCAT >>> To Unity
	nStatus BYTE: FROM Unity >>> TO TwinCAT	
	fTargetValue REAL: From TwinCAT >>> To Unity
	fActualValue REAL: FROM Unity >>> TO TwinCAT	
*)
FUNCTION_BLOCK FB_Drive EXTENDS FB_LinkDataREAL
VAR_INPUT
	nControl  		: BYTE;
	fTargetValue 	: REAL; //Target value to drive
END_VAR

VAR_OUTPUT
	nStatus  		: BYTE;
	fActualValue 	: REAL; //Actual value from drive
END_VAR

SUPER^();
Control := nControl;
ControlData := fTargetValue;
nStatus := Status;
fActualValue := StatusData;

END_FUNCTION_BLOCK

// Devices/Basic/FB_Lamp
(*
	Default Lamp device
*)
FUNCTION_BLOCK FB_Lamp EXTENDS FB_LinkDevice 
VAR_INPUT
	bEnable		: BOOL; //0-Lamp OFF, 1 - Lamp ON
END_VAR

SUPER^();
Control.0 := bEnable;

END_FUNCTION_BLOCK

// Devices/Basic/FB_Lock
(*
	Default Lock device
*)
FUNCTION_BLOCK FB_Lock EXTENDS FB_LinkDataByte 
VAR_INPUT
	bLock			: BOOL;
	nControlData	: BYTE;
END_VAR

VAR_OUTPUT	
	bClosed 		: BOOL;
	bLocked 		: BOOL; 
	nStatusData		: BYTE;
END_VAR

SUPER^();
Control.0 := bLock;
ControlData := nControlData;

bClosed := Status.0;
bLocked := Status.1;
nStatusData := StatusData;

END_FUNCTION_BLOCK

// Devices/Basic/FB_Panel
(*
	Basic panel with extended interface:
	nControl BYTE: From TwinCAT >>> To Unity
	nStatus BYTE: FROM Unity >>> TO TwinCAT	
	nControlData DWORD: From TwinCAT >>> To Unity
	nStatusData DWORD: FROM Unity >>> TO TwinCAT	
*)
FUNCTION_BLOCK FB_Panel EXTENDS FB_LinkDataDWord
VAR_INPUT
	nControlData  			: DWORD;
END_VAR

VAR_OUTPUT	
	nStatusData  			: DWORD;
END_VAR

SUPER^();
ControlData := nControlData;
nStatusData := StatusData;

END_FUNCTION_BLOCK

// Devices/Basic/FB_Reader
(*
	Default reader device	
*)
FUNCTION_BLOCK FB_Reader EXTENDS FB_LinkDataLWORD
VAR_INPUT
	nControl  		: BYTE;
	nCommand 		: ULINT; //Command ID
END_VAR

VAR_OUTPUT
	nStatus  		: BYTE;
	nResult			: ULINT; //Result Data
END_VAR

SUPER^();
Control := nControl;
ControlData := ULINT_TO_LWORD(nCommand);
nStatus := Status;
nResult := LWORD_TO_ULINT(StatusData);

END_FUNCTION_BLOCK

// Devices/Basic/FB_Robot
(*
	Default robot component with 12 axis interface	
*)
FUNCTION_BLOCK FB_Robot EXTENDS FB_LinkDevice
VAR_INPUT
	nControl  			: BYTE;	
	aJointTarget 		: ARRAY[0..11] OF REAL;	
END_VAR

VAR_OUTPUT
	nStatus  			: BYTE;
	aJointStatus 		: ARRAY[0..11] OF REAL;
END_VAR

VAR
	{attribute 'simulation_interface'}
	JointStatus AT %I* 	: ARRAY[0..11] OF REAL;
	{attribute 'simulation_interface'}
	JointTarget AT %Q* 	: ARRAY[0..11] OF REAL;
	
	{attribute 'hide'}
	_adrData			: LWORD;
	{attribute 'hide'}
	_nDataLength 		: UDINT;	
END_VAR

SUPER^();

IF (_adrData <> 0) THEN	
	MEMCPY(ADR(aJointTarget), _adrData, _nDataLength);
END_IF

Control := nControl;
MEMCPY(ADR(JointTarget), ADR(aJointTarget), 12 * 4);
MEMCPY(ADR(aJointStatus), ADR(JointStatus), 12 * 4);
nStatus := Status;

(*
	Assign the joint memory area for cyclic data exchange
*)
METHOD ConnectJoints : BOOL
VAR_INPUT
	Joints : ANY; //Adress to joints memmory area
	nJointCount : UDINT; //Number of joints
END_VAR
_adrData := Joints.pValue;
_nDataLength := LIMIT(0, nJointCount * 4, 12 * 4);
END_METHOD

METHOD INTERNAL GetJointsTarget : ARRAY[0..11] OF REAL;
GetJointsTarget := JointTarget;
END_METHOD

METHOD INTERNAL SetJointsStatus : BOOL
VAR_INPUT
	aJointsStatus : ARRAY[0..11] OF REAL;
END_VAR
JointStatus := aJointsStatus;
END_METHOD

END_FUNCTION_BLOCK

// Devices/Basic/FB_SensorAnalog
(*
	Default analog sensor device. 
	The stConfig structure is used to configure the scaling factor for transforming values into real-world units.
*)
FUNCTION_BLOCK FB_SensorAnalog EXTENDS FB_LinkDataReal 
VAR_INPUT
	nControl  		: BYTE;
	stConfig		: ST_ScaleConfig;
END_VAR

VAR_OUTPUT	
	nStatus  		: BYTE;
	nValue			: UINT;
	fValue			: REAL;
END_VAR

SUPER^();
Control := nControl;
fValue := StatusData;
nValue := LREAL_TO_UINT(F_ScaleLREAL(fValue, stConfig.fInputMin, stConfig.fInputMax, stConfig.fOutputMin, stConfig.fOutputMax));
nStatus := Status;

END_FUNCTION_BLOCK

// Devices/Basic/FB_SensorBinary
(*
	Default binary sensor device.
*)
FUNCTION_BLOCK FB_SensorBinary EXTENDS FB_LinkDevice 
VAR_OUTPUT
	bValue		: BOOL; 
END_VAR

SUPER^();
bValue := Status.0;

END_FUNCTION_BLOCK

// Devices/Basic/FB_Switch
(*
	Default switch device. 	
*)
FUNCTION_BLOCK FB_Switch EXTENDS FB_LinkDevice
VAR_INPUT		
	nControl  			: BYTE;
END_VAR

VAR_OUTPUT
	nStatus  			: BYTE;
END_VAR

SUPER^();
Control := nControl;
nStatus := Status;

END_FUNCTION_BLOCK

// Common/System/GVL_Core/fbSystem
PROPERTY PUBLIC fbSystem : REFERENCE TO FB_System
END_PROPERTY
